// TIA Portal project "2M - 1" (V16)

(* hardware
DEVICE "S7-1200 station_1"  S7-1200 Station
   slot 0: "Rack_0"  S7-1200 Rack  Rack  V1.0
   slot 1: "PLC_1"  CPU 1212C AC/DC/Rly  6ES7 212-1BE40-0XB0  V4.0
*)

// ===== PLC "PLC_1"  CPU 1212C AC/DC/Rly =====

VAR_GLOBAL   // PLC tag table "Default tag table"
   "start1" AT %I0.2 : Bool;
   "K1" AT %Q0.0 : Bool;
   "stop1" AT %I0.4 : Bool;
   "k2" AT %Q0.1 : Bool;
   "T1 tag" AT %M0.0 : Bool;
   "X" AT %M0.2 : Bool;
   "K3 RED" AT %Q0.2 : Bool;
   "Tag_1" AT %M1.0 : Bool;
   "Tag_2" AT %M3.2 : Bool;
   "STOP" AT %I0.3 : Bool;
   "Tag_3" AT %I0.5 : Bool;
   "Tag_4" AT %M4.0 : Bool;
END_VAR

// folder: System blocks/Program resources

DATA_BLOCK "T2"   // DB1
{ S7_Optimized_Access := 'TRUE' }
AUTHOR : Simatic
FAMILY : IEC
NAME : IEC_TMR
VERSION : 1.0
// stored: InstanceOfName IEC_TIMER
"IEC_TIMER"
BEGIN
END_DATA_BLOCK

DATA_BLOCK "T1"   // DB2
{ S7_Optimized_Access := 'TRUE' }
AUTHOR : Simatic
FAMILY : IEC
NAME : IEC_TMR
VERSION : 1.0
// stored: InstanceOfName IEC_TIMER
"IEC_TIMER"
BEGIN
END_DATA_BLOCK

DATA_BLOCK "counter1"   // DB3
{ S7_Optimized_Access := 'TRUE' }
AUTHOR : Simatic
FAMILY : IEC
NAME : CNTR
VERSION : 1.0
// stored: InstanceOfName IEC_COUNTER
"IEC_COUNTER"
BEGIN
END_DATA_BLOCK

// folder: (top level)

ORGANIZATION_BLOCK "Main"   // OB1, LAD, ProgramCycle
TITLE = "Main Program Sweep (Cycle)"
{ S7_Optimized_Access := 'TRUE' }
VERSION : 0.1
   VAR_INPUT
      Initial_Call : Bool;   // Initial call of this OB
      Remanence : Bool;   // =True, if remanent data are available
   END_VAR
BEGIN

REGION Network 1: start
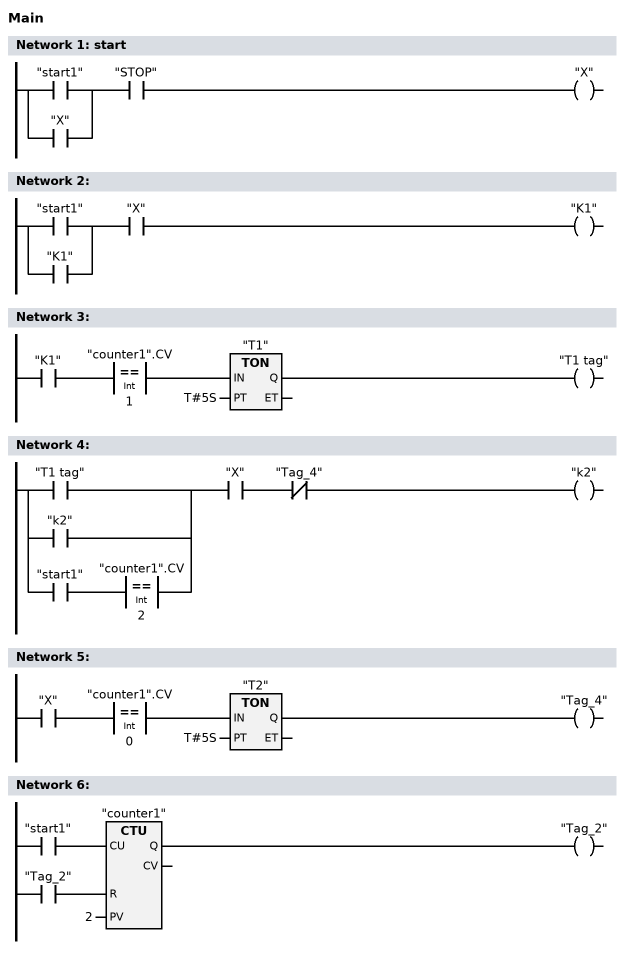
   RUNG wire#powerrail
      Contact( "start1" )
      wire#w1
      Contact( "STOP" )
      Coil( "X" )
   END_RUNG
   RUNG wire#powerrail
      Contact( "X" )
   END_RUNG wire#w1
   // the same network as SCL:
   "X" := ("start1" OR "X") AND "STOP";
END_REGION

REGION Network 2
   RUNG wire#powerrail
      Contact( "start1" )
      wire#w1
      Contact( "X" )
      Coil( "K1" )
   END_RUNG
   RUNG wire#powerrail
      Contact( "K1" )
   END_RUNG wire#w1
   // the same network as SCL:
   "K1" := ("start1" OR "K1") AND "X";
END_REGION

REGION Network 3
   "T1".TON(IN := "K1" AND ("counter1".CV = 1), PT := T#5S);
   "T1 tag" := "T1".Q;
END_REGION

REGION Network 4
   RUNG wire#powerrail
      Contact( "T1 tag" )
      wire#w1
      Contact( "X" )
      I_Contact( "Tag_4" )
      Coil( "k2" )
   END_RUNG
   RUNG wire#powerrail
      Contact( "k2" )
   END_RUNG wire#w1
   RUNG wire#powerrail
      Contact( "start1" )
      { S7_Templates := "SrcType := Int" } EQ_Contact(in1 := "counter1".CV, in2 := 2)
   END_RUNG wire#w1
   // the same network as SCL:
   "k2" := ("T1 tag" OR "k2" OR ("start1" AND ("counter1".CV = 2))) AND "X" AND NOT "Tag_4";
END_REGION

REGION Network 5
   "T2".TON(IN := "X" AND ("counter1".CV = 0), PT := T#5S);
   "Tag_4" := "T2".Q;
END_REGION

REGION Network 6
   "counter1".CTU(CU := "start1", R := "Tag_2", PV := 2);
   "Tag_2" := "counter1".Q;
END_REGION
END_ORGANIZATION_BLOCK